{attribute addProperty BoxType "EL3314-0090-0016"}
{attribute addProperty Id "StatusAT %I*Status_F0C7FE3C1621ValueAT %I*INT16217"}
{attribute addProperty CRC "4050261517"}
{attribute addProperty SizeInBites "32"}
{attribute addProperty SizeInBytes "4"}
TYPE TC_Inputs_Channel_F16A160D :
STRUCT
	{attribute addProperty Name "Status"}
	Status AT %I* : Status_F0C7FE3C;
	{attribute addProperty Name "Value"}
	Value AT %I* : INT;
END_STRUCT
END_TYPE

(* stored: Version 1.2.0.0, ProductVersion 3.1.4024.9
   DUT TC_Inputs_Channel_F16A160D: Id {1bcc8087-e933-433c-a3bc-040a8f41defa} *)
